// SIMATIC S7-200 project (STEP 7-Micro/WIN), CPU 221 REL 01.10

ORGANIZATION_BLOCK 主程序:OB1
TITLE=程序注释
BEGIN
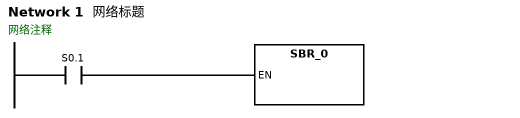
Network 1 // 网络标题
// 网络注释
LD     S0.1
CALL   SBR_0:SBR0
END_ORGANIZATION_BLOCK

SUBROUTINE_BLOCK SBR_0:SBR0
TITLE=程序注释
BEGIN
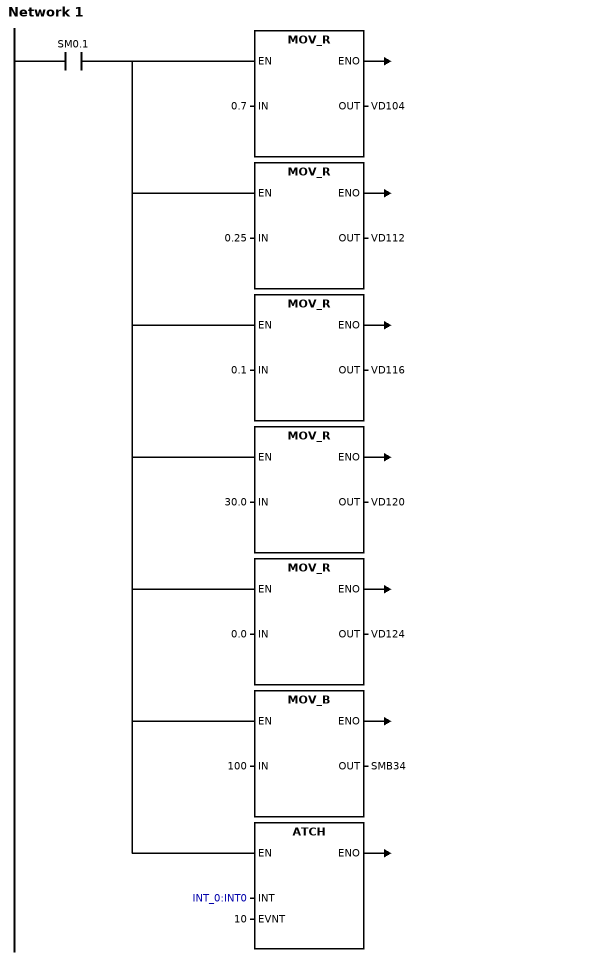
Network 1
LD     SM0.1
MOVR   0.7, VD104
MOVR   0.25, VD112
MOVR   0.1, VD116
MOVR   30.0, VD120
MOVR   0.0, VD124
MOVB   100, SMB34
ATCH   INT_0:INT0, 10
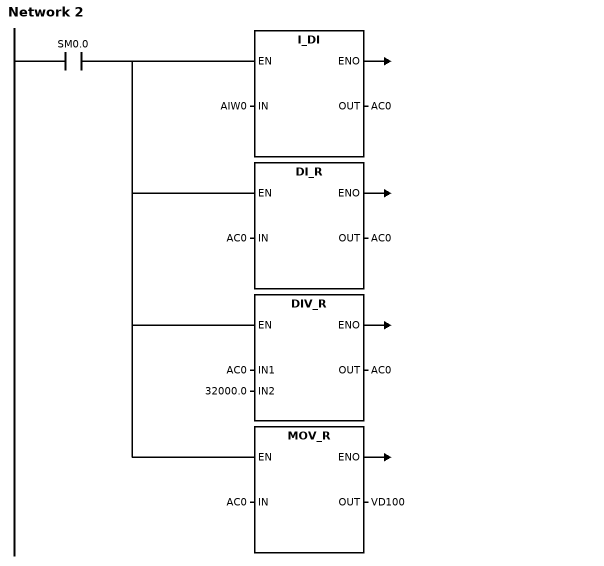
Network 2
LD     SM0.0
ITD    AIW0, AC0
DTR    AC0, AC0
/R     32000.0, AC0
MOVR   AC0, VD100
Network 25 // 网络标题
// 网络注释
END_SUBROUTINE_BLOCK
